PROGRAM p_task2
VAR
END_VAR

END_PROGRAM

(* stored: Version 1.1.0.1, ProductVersion 3.1.4024.12
   POU p_task2: Id {ddb7acdb-c93a-4bb6-9952-7918696a7e26}, SpecialFunc None *)
